(* IEC 61131-3 sources: Industry-PLC-LLM/data/PLCBEAD_repo/PLCBEAD_PLCEmbed-main/PLC-BEAD/Source/GEB/GDF, 1 file *)

(* ---- GDF.ST ---- *)
FUNCTION GDF:REAL

	VAR_INPUT
		X :	REAL;
	END_VAR

	IF X = 0.0 THEN
		GDF := 0.0;
	ELSIF X > 15.0 THEN
		GDF := 1.5707963267949;
	ELSIF X < -15.0 THEN
		GDF := -1.5707963267949;
	ELSE
		GDF := ATAN(EXP(X)) * 2.0 - 1.5707963267949;
	END_IF;

END_FUNCTION

PROGRAM program0
  VAR
    X :	REAL;
    LocalOUT  : REAL;
  END_VAR

  LocalOUT := GDF(X);
END_PROGRAM
